PROGRAM MAIN
VAR
END_VAR

END_PROGRAM

(* stored: Version 1.1.0.1
   POU MAIN: Id {fbf91538-5e12-4536-b105-9f5441ce8fb4} *)
